FUNCTION_BLOCK Seq_Ausrichten_Plates EXTENDS FB_Basis IMPLEMENTS I_Sequenz
VAR_INPUT
	// Skillzuweisung
	R_Move			:I_Skill_RoboterErweitert;
	
	// Prozessparameter		
	RobParam				:ARRAY[0..4] OF sRoboterProzessVariablen;
	ErreichtParam			:sKraftVariablen;
END_VAR
VAR_OUTPUT
END_VAR
VAR
	ErreichtParamReset		:sKraftVariablen;
END_VAR

// Ablauf
ACT_Ablauf();

// Zustandshandling
CASE iState OF
	0:	// BEREIT
		IF bStart THEN
			bStart := FALSE;
			iState := 1;
		END_IF
	1:	// LAUFEND
		IF eSysCommand = 4 THEN
			bReset := TRUE;
			SFCReset := TRUE;
		END_IF
		
		IF bBeendet OR bReset THEN
			bReset := FALSE;
			SFCReset := FALSE;
			iState := 0;
		END_IF
END_CASE

ACTION ACT_1:
R_Move.P_RobotParam := RobParam[0];
END_ACTION

ACTION ACT_2:
R_Move.P_RobotParam := RobParam[1];
END_ACTION

ACTION ACT_3:
R_Move.P_RobotParam := RobParam[2];
R_Move.P_Erreicht := ErreichtParam;
END_ACTION

ACTION ACT_4:
R_Move.P_RobotParam := RobParam[3];
END_ACTION

ACTION ACT_5:
R_Move.P_RobotParam := RobParam[4];
END_ACTION

ACTION ACT_Ablauf:
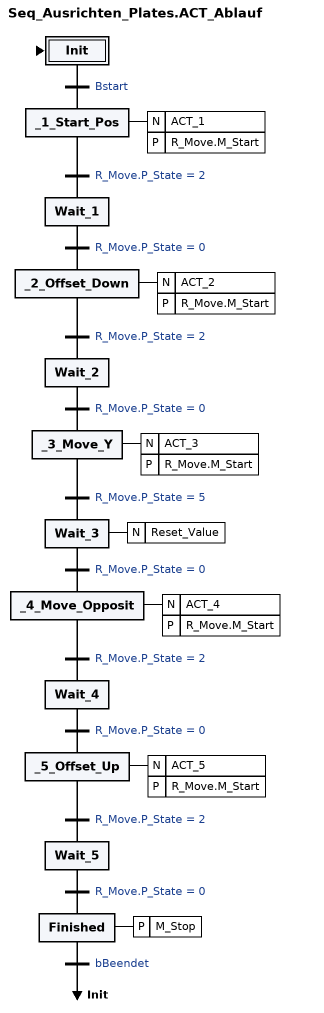
INITIAL_STEP Init:
END_STEP
TRANSITION FROM Init TO _1_Start_Pos
    := Bstart;
END_TRANSITION
STEP _1_Start_Pos:
    ACT_1(N);
    R_Move.M_Start(P);
END_STEP
TRANSITION FROM _1_Start_Pos TO Wait_1
    := R_Move.P_State = 2;
END_TRANSITION
STEP Wait_1:
END_STEP
TRANSITION FROM Wait_1 TO _2_Offset_Down
    := R_Move.P_State = 0;
END_TRANSITION
STEP _2_Offset_Down:
    ACT_2(N);
    R_Move.M_Start(P);
END_STEP
TRANSITION FROM _2_Offset_Down TO Wait_2
    := R_Move.P_State = 2;
END_TRANSITION
STEP Wait_2:
END_STEP
TRANSITION FROM Wait_2 TO _3_Move_Y
    := R_Move.P_State = 0;
END_TRANSITION
STEP _3_Move_Y:
    ACT_3(N);
    R_Move.M_Start(P);
END_STEP
TRANSITION FROM _3_Move_Y TO Wait_3
    := R_Move.P_State = 5;
END_TRANSITION
STEP Wait_3:
    Reset_Value(N);
END_STEP
TRANSITION FROM Wait_3 TO _4_Move_Opposit
    := R_Move.P_State = 0;
END_TRANSITION
STEP _4_Move_Opposit:
    ACT_4(N);
    R_Move.M_Start(P);
END_STEP
TRANSITION FROM _4_Move_Opposit TO Wait_4
    := R_Move.P_State = 2;
END_TRANSITION
STEP Wait_4:
END_STEP
TRANSITION FROM Wait_4 TO _5_Offset_Up
    := R_Move.P_State = 0;
END_TRANSITION
STEP _5_Offset_Up:
    ACT_5(N);
    R_Move.M_Start(P);
END_STEP
TRANSITION FROM _5_Offset_Up TO Wait_5
    := R_Move.P_State = 2;
END_TRANSITION
STEP Wait_5:
END_STEP
TRANSITION FROM Wait_5 TO Finished
    := R_Move.P_State = 0;
END_TRANSITION
STEP Finished:
    M_Stop(P);
END_STEP
TRANSITION FROM Finished TO Init
    := bBeendet;
END_TRANSITION
END_ACTION

ACTION Reset_Value:
ErreichtParamReset.Fx := 0;
ErreichtParamReset.Fy := 0;
ErreichtParamReset.Fz := 0;

R_Move.P_Erreicht := ErreichtParamReset;
END_ACTION

END_FUNCTION_BLOCK

(* stored: Version 1.1.0.1
   POU Seq_Ausrichten_Plates: Id {f93ae988-edc6-473e-8267-149d415ff47f}, SpecialFunc None
   Folder 01_Zuweisung: Id {7abb2af8-3692-49fa-8ae7-84439d381ae9}
   Action ACT_1: Id {e21f4808-1d84-4ece-ac6e-8ecf7bac585f}
   Action ACT_2: Id {186cb54d-aba8-4453-b5c3-f5d583bba9be}
   Action ACT_3: Id {dc6ebae0-2090-46c0-9e84-96aa41fbabfc}
   Action ACT_4: Id {62177a7d-cedd-44d6-96f4-b7ee8dd0099c}
   Action ACT_5: Id {31aa8d9d-24a4-4fec-8279-bc82c0b84323}
   Action ACT_Ablauf: Id {00d5be4d-f48d-4a1b-97c3-f9006e20d8b0}
   Action Reset_Value: Id {011cffe1-d850-4451-b57f-d87f1248d423} *)
